ABB RAPID module: Module1.mod

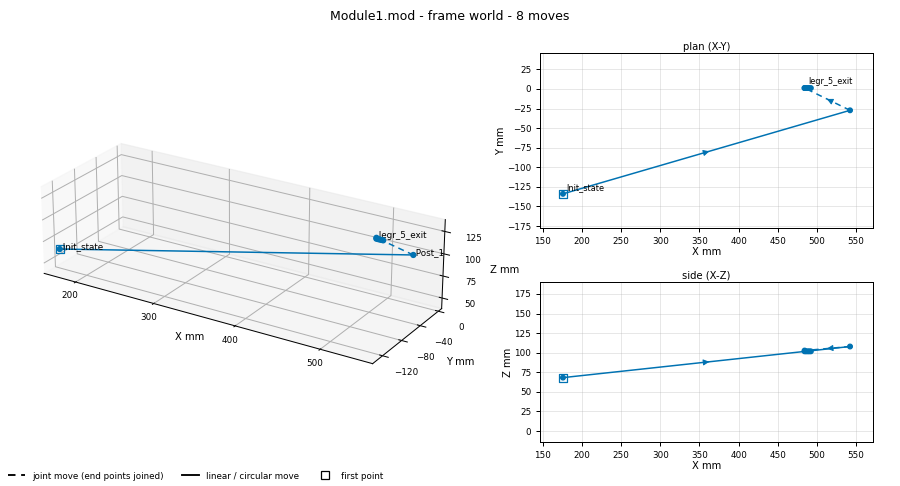
[picture p0: tool path of Module1.mod in frame world, 8 of 8 moves have a stored position in this frame; points joined in program order, loops and branches not executed]
MODULE Module1
        CONST robtarget Init_state:=[[175.771799788,-133.936334157,68.163208612],[0.220019445,-0.124834347,0.967057146,0.028430707],[0,0,-2,4],[-101.964427132,9E+09,9E+09,9E+09,9E+09,9E+09]];
    CONST robtarget Post_1:=[[542.319387186,-27.270592964,107.891310148],[0.380274295,0.087924872,0.895606571,0.213423401],[1,1,-2,4],[-171.216572779,9E+09,9E+09,9E+09,9E+09,9E+09]];
    CONST robtarget legr_5_exit:=[[484.286991076,1.172337286,102.734659718],[0.381901533,0.089000385,0.894935668,0.21288565],[1,2,-2,4],[124.109986755,9E+09,9E+09,9E+09,9E+09,9E+09]];
    CONST robtarget Welding_legr_1:=[[488.28569584,1.174716546,101.736284395],[0.381903905,0.089001119,0.894934472,0.212886116],[1,2,-2,4],[124.109990085,9E+09,9E+09,9E+09,9E+09,9E+09]];
    CONST robtarget Welding_legr_2:=[[490.285916331,1.174333865,101.735976988],[0.381903397,0.089000929,0.894934769,0.21288586],[1,2,-2,4],[124.10999081,9E+09,9E+09,9E+09,9E+09,9E+09]];
    CONST robtarget Welding_legr_3:=[[492.28611356,1.174026671,101.735814814],[0.381903161,0.089000873,0.894934883,0.212885827],[1,2,-2,4],[124.109989426,9E+09,9E+09,9E+09,9E+09,9E+09]];
    CONST robtarget Welding_legr_4:=[[486.286692413,1.172930738,101.734952345],[0.381902109,0.089000616,0.894935318,0.212885992],[1,2,-2,4],[124.109983855,9E+09,9E+09,9E+09,9E+09,9E+09]];
    CONST robtarget Welding_legr_5:=[[484.286867502,1.172484711,101.734755535],[0.38190173,0.08900051,0.894935551,0.212885737],[1,2,-2,4],[124.109987599,9E+09,9E+09,9E+09,9E+09,9E+09]];
!***********************************************************
    !
    ! Module:  Module1
    !
    ! Description:
    !   <Insert description here>
    !
    ! Author: mmora
    !
    ! Version: 1.0
    !
    !***********************************************************


    !***********************************************************
    !
    ! Procedure main
    !
    !   This is the entry point of your program
    !
    !***********************************************************
    PROC main()
        !Add your code here
        MoveL Init_state,v200,fine,MyTool\WObj:=wobj0;
        MoveL Post_1,v200,fine,MyTool\WObj:=wobj0;
        MoveJ legr_5_exit,v200,fine,MyTool\WObj:=wobj0;
        MoveJ Welding_legr_1,v200,fine,MyTool\WObj:=wobj0;
        MoveJ Welding_legr_2,v200,fine,MyTool\WObj:=wobj0;
        MoveJ Welding_legr_3,v200,fine,MyTool\WObj:=wobj0;
        MoveJ Welding_legr_4,v200,fine,MyTool\WObj:=wobj0;
        MoveJ Welding_legr_5,v200,fine,MyTool\WObj:=wobj0;
    ENDPROC
ENDMODULE
